(* IEC 61131-3 sources: CODESYS-IO-Visualization/CODESYS-IO-Visualization.fbsproj/Pi.device.xml.v3^/Plc Logic.plclogic.xml.v3^/Application.application.xml.v3^/Programs/4_Process, 1 file *)

(* ---- Main_Process.prg.st ---- *)
PROGRAM Main_Process

VAR
	Init: BOOL := TRUE;
END_VAR

IF Init THEN
	Site.Plant.Pump1.InletValve.HMI.SWITCH0[1] := 1;
	Site.Plant.Pump1.OutletValve.HMI.SWITCH0[1] := 1;
	Site.Plant.Pump1.InletValve.HMI.REAL0[20] := 100.0;
	Site.Plant.Pump1.OutletValve.HMI.REAL0[20] := 50.0;

	Site.Plant.Pump1.VFD.Remote := TRUE;

	Init := FALSE;
END_IF;

Process_RotorkValve_Auto(valve := Site.Plant.Pump1.InletValve);
Process_RotorkValve_Auto(valve := Site.Plant.Pump1.OutletValve);
Process_PumpVFD(equip := Site.Plant.Pump1.VFD);
